ABB RAPID module: Irc6UploadResult.mod

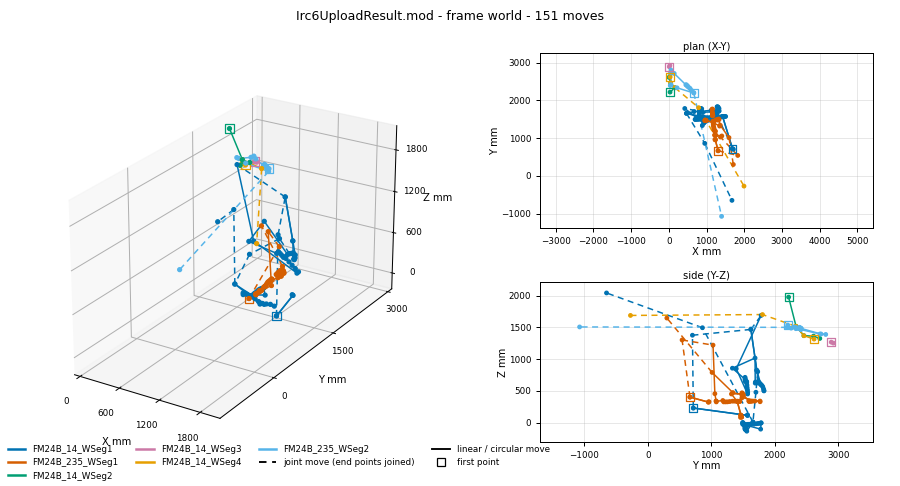
[picture p0: tool path of Irc6UploadResult.mod in frame world, 151 of 155 moves have a stored position in this frame; points joined in program order, loops and branches not executed]
%%%
  VERSION:1
  LANGUAGE:ENGLISH
%%%

MODULE FM24BSegment
!# Process Simulate on eMServer 14 to ABB Rapid Volvo download
!# ------------------------------------------------
!# CREATED   : 26/04/2018 16:18:21 by yogesha
!# CELL      : 2V3 Enginecase_V1
!# ROBOT     : AR21_IRB6700_220-265_SW_IRC5_Grey
!# PROGRAM   : FM24BSegment
!# VOLP      : Abb-Rapid-Volvo 3.14.1
!# RCS       : 6.04.irc5
!# CONTROLLER: 6.0 RW6


!# ----------------------------------------------
!# ------ ROBTARGET
!# ----------------------------------------------
  LOCAL CONST robtarget Towp429210G_10:=[[4329.26,-293.89,1820.66],[0.041749,0.120567,0.991812,0.005418],[-1,0,-1,0],[9e+09,300,9e+09,9e+09,9e+09,9e+09]];
  LOCAL CONST robtarget Towp429210G_20:=[[3458.99,-78.17,1742.31],[0.041752,0.120591,0.991809,0.005444],[0,1,-1,0],[9e+09,25,9e+09,9e+09,9e+09,9e+09]];
  LOCAL CONST robtarget wp429210G:=[[3458.44,-77.54,1729.33],[0.0417533,0.12059,0.991809,0.00543544],[-1,1,-1,0],[9E+09,24.9996,9E+09,9E+09,9E+09,9E+09]];
  LOCAL CONST robtarget Towp431238_10:=[[3458.99,-78.17,1742.31],[0.041752,0.12059,0.991809,0.005444],[0,1,-1,0],[9e+09,25,9e+09,9e+09,9e+09,9e+09]];
  LOCAL CONST robtarget Towp431238_20:=[[4329.31,-293.87,1820.63],[0.041749,0.120567,0.991812,0.005418],[-1,0,-1,0],[9e+09,300,9e+09,9e+09,9e+09,9e+09]];
  LOCAL CONST robtarget Towp431238_30:=[[4344.72,-1189.03,1103.91],[0.199902,-0.332679,-0.8027,-0.452809],[-1,0,-1,0],[9e+09,300,9e+09,9e+09,9e+09,9e+09]];
  LOCAL CONST robtarget Towp431238_40:=[[3393.84,-1017.32,754.57],[0.232734,-0.408546,-0.787878,-0.39771],[0,-1,0,0],[9e+09,200,9e+09,9e+09,9e+09,9e+09]];
  LOCAL CONST robtarget Towp431238_50:=[[3305.21,-568.3,1223.23],[0.212691,-0.544427,-0.755771,-0.295249],[0,-1,0,0],[9e+09,200,9e+09,9e+09,9e+09,9e+09]];
  LOCAL CONST robtarget Towp431238_60:=[[3241.28,-398.98,1372.39],[0.145145,-0.515318,-0.836002,-0.120336],[0,-1,0,0],[9E+09,110.437,9E+09,9E+09,9E+09,9E+09]];
  LOCAL CONST robtarget Towp431238_70:=[[3190.42,-299.46,1405.89],[0.0308017,-0.526819,-0.84797,-0.0495987],[0,0,0,0],[9E+09,44.8475,9E+09,9E+09,9E+09,9E+09]];
  LOCAL CONST robtarget wp431238:=[[3189.5,-297.98,1394.24],[0.030797,-0.526829,-0.847965,-0.049568],[0,0,0,0],[9E+09,24.9996,9E+09,9E+09,9E+09,9E+09]];
  LOCAL CONST robtarget wp429282:=[[3210,-357.62,1373.29],[0.141617,-0.469636,-0.834318,-0.251596],[0,-1,0,0],[9E+09,24.9981,9E+09,9E+09,9E+09,9E+09]];
  LOCAL CONST robtarget wp429283G:=[[3224.18,-374.72,1360.26],[0.231783,-0.536585,-0.744868,-0.321753],[0,-1,0,0],[9E+09,25.0004,9E+09,9E+09,9E+09,9E+09]];
  LOCAL CONST robtarget wp429284:=[[3247.29,-390.89,1343.19],[0.335931,-0.549838,-0.652262,-0.399229],[0,-1,1,0],[9E+09,24.9981,9E+09,9E+09,9E+09,9E+09]];
  LOCAL CONST robtarget wp429285:=[[3274.81,-399.51,1329.50],[0.386439,-0.541317,-0.588631,-0.459515],[0,-1,1,0],[9E+09,24.9999,9E+09,9E+09,9E+09,9E+09]];
  LOCAL CONST robtarget Towp429203G_10:=[[3268.63,-416.83,1335.22],[0.354523,-0.56273,-0.614198,-0.424746],[0,-1,1,0],[9e+09,150,9e+09,9e+09,9e+09,9e+09]];
  LOCAL CONST robtarget Towp429203G_20:=[[3305.16,-568.32,1223.25],[0.212691,-0.544427,-0.755771,-0.295249],[0,-1,0,0],[9e+09,150,9e+09,9e+09,9e+09,9e+09]];
  LOCAL CONST robtarget Towp429203G_30:=[[3393.84,-1017.32,754.57],[0.232734,-0.408546,-0.787878,-0.39771],[0,-1,0,0],[9e+09,150,9e+09,9e+09,9e+09,9e+09]];
  LOCAL CONST robtarget Towp429203G_40:=[[3171.33,-657.72,-21.12],[0.192002,0.140607,-0.823074,0.515668],[0,-1,-2,0],[9e+09,270,9e+09,9e+09,9e+09,9e+09]];
  LOCAL CONST robtarget Towp429203G_50:=[[3598.53,-315.02,877.27],[0.496486,0.441662,-0.526165,0.530647],[0,-1,-2,0],[9e+09,270,9e+09,9e+09,9e+09,9e+09]];
  LOCAL CONST robtarget Towp429203G_60:=[[3461.55,-373.9,1571.05],[0.496488,0.441684,-0.526144,0.530648],[0,-1,-2,0],[9e+09,270,9e+09,9e+09,9e+09,9e+09]];
  LOCAL CONST robtarget wp429203G:=[[3461.52,-406.31,1573.04],[0.496495,0.441685,-0.526141,0.530644],[0,-1,-2,0],[9E+09,24.9993,9E+09,9E+09,9E+09,9E+09]];
  LOCAL CONST robtarget wp429202:=[[3461.25,-404.66,1511.75],[0.423916,0.425319,-0.564527,0.566311],[0,0,-2,0],[9E+09,25.0001,9E+09,9E+09,9E+09,9E+09]];
  LOCAL CONST robtarget wp429201:=[[3462.97,-404.15,1452.61],[0.449062,0.449065,-0.546205,0.546209],[0,-1,-2,0],[9E+09,25.0001,9E+09,9E+09,9E+09,9E+09]];
  LOCAL CONST robtarget wp429200:=[[3463.05,-405.21,1392.26],[0.449062,0.449063,-0.546207,0.546209],[0,-1,-2,0],[9E+09,24.9996,9E+09,9E+09,9E+09,9E+09]];
  LOCAL CONST robtarget wp429199:=[[3463.42,-406.70,1332.03],[0.444279,0.444281,-0.550103,0.550107],[0,-1,-2,0],[9E+09,25.0001,9E+09,9E+09,9E+09,9E+09]];
  LOCAL CONST robtarget wp432680G:=[[3461.83,-405.59,1302.23],[0.407023,0.377506,-0.565637,0.609817],[0,0,-2,0],[9E+09,25.0011,9E+09,9E+09,9E+09,9E+09]];
  LOCAL CONST robtarget wp429273:=[[3482.99,-404.27,1300.72],[0.483124,0.448113,-0.511515,0.551488],[0,0,-2,0],[9E+09,25.0001,9E+09,9E+09,9E+09,9E+09]];
  LOCAL CONST robtarget wp429272:=[[3482.16,-405.26,1268.30],[0.399742,0.399756,-0.583268,0.583267],[0,0,-2,0],[9E+09,24.9996,9E+09,9E+09,9E+09,9E+09]];
  LOCAL CONST robtarget wp429271:=[[3481.99,-406.34,1234.52],[0.399739,0.399755,-0.583271,0.583267],[0,0,-2,0],[9E+09,24.9996,9E+09,9E+09,9E+09,9E+09]];
  LOCAL CONST robtarget wp429270G:=[[3482.14,-406.55,1199.88],[0.373924,0.373932,-0.600148,0.600148],[0,0,-2,0],[9E+09,25.0001,9E+09,9E+09,9E+09,9E+09]];
  LOCAL CONST robtarget Towp429287_10:=[[3479.92,-364.68,1199.99],[0.373918,0.3739,-0.600176,0.600144],[0,0,-2,0],[9e+09,200,9e+09,9e+09,9e+09,9e+09]];
  LOCAL CONST robtarget Towp429287_20:=[[3656.14,-294.7,840.95],[0.373913,0.37388,-0.600196,0.600139],[0,0,-2,0],[9e+09,225,9e+09,9e+09,9e+09,9e+09]];
  LOCAL CONST robtarget Towp429287_30:=[[3301.96,-446.59,772.7],[0.485357,0.438793,-0.503692,0.564078],[0,0,-2,0],[9e+09,100,9e+09,9e+09,9e+09,9e+09]];
  LOCAL CONST robtarget Towp429287_40:=[[3325.47,-372.58,1301.67],[0.485362,0.438786,-0.503693,0.564077],[0,0,-2,0],[9E+09,99.9999,9E+09,9E+09,9E+09,9E+09]];
  LOCAL CONST robtarget wp429287:=[[3324.91,-401.60,1310.54],[0.485353,0.438798,-0.503689,0.564081],[0,0,-2,0],[9E+09,24.9997,9E+09,9E+09,9E+09,9E+09]];
  LOCAL CONST robtarget wp429286:=[[3296.51,-398.64,1318.97],[0.533282,0.418254,-0.478916,0.557955],[0,0,-2,0],[9E+09,24.9994,9E+09,9E+09,9E+09,9E+09]];
  LOCAL CONST robtarget Towp429216G_10:=[[3297.45,-384.27,1310.22],[0.533276,0.418255,-0.478914,0.557961],[0,0,-2,0],[9e+09,100,9e+09,9e+09,9e+09,9e+09]];
  LOCAL CONST robtarget Towp429216G_20:=[[3275.54,-416.71,1074.85],[0.513983,0.427519,-0.492769,0.556981],[0,0,-2,0],[9E+09,100,9E+09,9E+09,9E+09,9E+09]];
  LOCAL CONST robtarget Towp429216G_30:=[[3302.69,609.90,1079.32],[0.491897,0.48192,-0.351229,0.634373],[1,0,-1,0],[9E+09,200,9E+09,9E+09,9E+09,9E+09]];
  LOCAL CONST robtarget Towp429216G_40:=[[3432.85,433.93,1516.60],[0.368379,0.736883,-0.491235,0.282824],[1,-1,-1,0],[9E+09,140.674,9E+09,9E+09,9E+09,9E+09]];
  LOCAL CONST robtarget wp429216G:=[[3460.36,263.26,1671.83],[0.365723,0.756894,-0.437503,0.319295],[1,-1,-1,0],[9E+09,25.0001,9E+09,9E+09,9E+09,9E+09]];
  LOCAL CONST robtarget wp429217:=[[3460.06,290.30,1618.13],[0.33206,0.726093,-0.53763,0.271071],[1,-1,-1,0],[9E+09,24.9996,9E+09,9E+09,9E+09,9E+09]];
  LOCAL CONST robtarget wp429218:=[[3460.14,334.70,1576.96],[0.2765,0.779954,-0.522201,0.206218],[1,-1,-1,0],[9E+09,25.0001,9E+09,9E+09,9E+09,9E+09]];
  LOCAL CONST robtarget wp429219:=[[3461.00,376.35,1534.46],[0.388866,0.719255,-0.497691,0.289411],[1,-1,-1,0],[9E+09,25.0001,9E+09,9E+09,9E+09,9E+09]];
  LOCAL CONST robtarget wp429220G:=[[3462.24,400.89,1481.39],[0.481708,0.646297,-0.461703,0.370253],[1,-1,-1,0],[9E+09,25.0001,9E+09,9E+09,9E+09,9E+09]];
  LOCAL CONST robtarget wp429221:=[[3462.42,411.51,1422.21],[0.547313,0.587418,-0.431084,0.41177],[1,-1,-1,0],[9E+09,25.0001,9E+09,9E+09,9E+09,9E+09]];
  LOCAL CONST robtarget wp429222:=[[3462.28,413.55,1392.21],[0.582433,0.580357,-0.398114,0.40677],[1,-1,-1,0],[9E+09,25.0001,9E+09,9E+09,9E+09,9E+09]];
  LOCAL CONST robtarget wp431518G:=[[3458.41,420.46,1359.28],[0.377325,0.73689,-0.499266,0.255641],[1,-1,-1,0],[9E+09,25.0001,9E+09,9E+09,9E+09,9E+09]];
  LOCAL CONST robtarget wp429263:=[[3481.41,418.56,1361.00],[0.373199,0.728795,-0.510991,0.261665],[1,-1,-1,0],[9E+09,25.0001,9E+09,9E+09,9E+09,9E+09]];
  LOCAL CONST robtarget wp429264:=[[3481.76,433.47,1336.37],[0.467923,0.686198,-0.460136,0.313775],[1,-1,-1,0],[9E+09,25.0001,9E+09,9E+09,9E+09,9E+09]];
  LOCAL CONST robtarget wp429265:=[[3483.02,442.45,1306.90],[0.514146,0.672387,-0.422993,0.32346],[1,-1,-1,0],[9E+09,25.0001,9E+09,9E+09,9E+09,9E+09]];
  LOCAL CONST robtarget wp429266:=[[3481.16,455.69,1277.06],[0.34984,0.757592,-0.500294,0.231024],[1,-1,-1,0],[9E+09,25.0001,9E+09,9E+09,9E+09,9E+09]];
  LOCAL CONST robtarget wp429267G:=[[3480.50,478.18,1255.11],[0.355857,0.777298,-0.471735,0.215962],[1,-1,-1,0],[9E+09,24.9996,9E+09,9E+09,9E+09,9E+09]];
  LOCAL CONST robtarget Towp433102G_10:=[[3479.99,496.17,1270.97],[0.355865,0.777283,-0.471751,0.215968],[1,-1,-1,0],[9e+09,150,9e+09,9e+09,9e+09,9e+09]];
  LOCAL CONST robtarget Towp433102G_20:=[[3211.27,432.33,1467.96],[0.202641,0.500327,-0.809314,0.231561],[1,-1,0,0],[9e+09,130,9e+09,9e+09,9e+09,9e+09]];
  LOCAL CONST robtarget wp433102G:=[[3202.22,373.10,1382.13],[0.131743,0.518539,-0.82381,0.187345],[1,-1,0,0],[9E+09,25.0006,9E+09,9E+09,9E+09,9E+09]];
  LOCAL CONST robtarget Towp429230_10:=[[3202.31,375.23,1386.42],[0.138512,0.516986,-0.822694,0.19161],[1,-1,0,0],[9e+09,25,9e+09,9e+09,9e+09,9e+09]];
  LOCAL CONST robtarget wp429230:=[[3222.80,391.61,1372.68],[0.177635,0.590788,-0.753609,0.226912],[1,-1,0,0],[9E+09,24.9996,9E+09,9E+09,9E+09,9E+09]];
  LOCAL CONST robtarget wp429229:=[[3247.09,402.51,1364.21],[0.258409,0.688458,-0.63409,0.239124],[1,-1,-1,0],[9E+09,25.0001,9E+09,9E+09,9E+09,9E+09]];
  LOCAL CONST robtarget wp429228:=[[3274.77,411.27,1360.35],[0.299271,0.704832,-0.591093,0.25349],[1,-1,-1,0],[9E+09,24.9994,9E+09,9E+09,9E+09,9E+09]];
  LOCAL CONST robtarget wp435330:=[[3311.15,418.41,1362.24],[0.319174,0.778948,-0.441981,0.309873],[1,-1,-1,0],[9E+09,24.9999,9E+09,9E+09,9E+09,9E+09]];
  LOCAL CONST robtarget wp429225:=[[3360.20,420.14,1361.29],[0.37043,0.735721,-0.506434,0.254992],[1,-1,-1,0],[9E+09,25.0001,9E+09,9E+09,9E+09,9E+09]];
  LOCAL CONST robtarget wp429224:=[[3388.55,420.54,1361.74],[0.369194,0.732673,-0.510579,0.257285],[1,-1,-1,0],[9E+09,24.9981,9E+09,9E+09,9E+09,9E+09]];
  LOCAL CONST robtarget wp429223:=[[3418.13,420.96,1362.93],[0.373371,0.733676,-0.505974,0.257495],[1,-1,-1,0],[9E+09,24.9999,9E+09,9E+09,9E+09,9E+09]];
  LOCAL CONST robtarget Frwp429223_10:=[[3419.47,437.29,1376.00],[0.37778,0.742391,-0.493107,0.250966],[1,-1,-1,0],[9E+09,150,9E+09,9E+09,9E+09,9E+09]];
  LOCAL CONST robtarget Frwp429223_20:=[[3302.73,609.92,1079.3],[0.566533,0.521636,-0.288972,0.568711],[1,0,-1,0],[9e+09,200,9e+09,9e+09,9e+09,9e+09]];
  LOCAL CONST robtarget Frwp429223_30:=[[4131.69,-803.62,455.75],[0.261761,0.576711,-0.326948,0.70142],[1,-1,-1,0],[9E+09,330,9E+09,9E+09,9E+09,9E+09]];
  LOCAL CONST robtarget Frwp429223_40:=[[5691.66,-1613.7,572.8],[0.123608,0.891176,-0.221992,0.375828],[0,-1,-2,0],[9e+09,50,9e+09,9e+09,9e+09,9e+09]];
  LOCAL CONST robtarget Towp431451G_10:=[[4354.11,-179.99,1414.82],[0.017246,-0.153263,-0.988031,-0.002663],[-1,0,-1,0],[9e+09,50,9e+09,9e+09,9e+09,9e+09]];
  LOCAL CONST robtarget Towp431451G_20:=[[4058.85,-86.14,1425.65],[0.017246,-0.153263,-0.988031,-0.002663],[-1,0,-1,0],[9e+09,50,9e+09,9e+09,9e+09,9e+09]];
  LOCAL CONST robtarget wp431451G:=[[4047.79,-84.24,1413.94],[0.0172455,-0.153278,-0.988029,-0.00267298],[-1,0,-1,0],[9E+09,24.9999,9E+09,9E+09,9E+09,9E+09]];
  LOCAL CONST robtarget Towp431454_10:=[[4058.85,-86.14,1425.65],[0.017247,-0.153263,-0.988031,-0.002663],[-1,0,-1,0],[9e+09,50,9e+09,9e+09,9e+09,9e+09]];
  LOCAL CONST robtarget Towp431454_20:=[[4354.11,-179.99,1414.82],[0.017247,-0.153263,-0.988031,-0.002663],[-1,0,-1,0],[9e+09,50,9e+09,9e+09,9e+09,9e+09]];
  LOCAL CONST robtarget Towp431454_30:=[[4515.84,-1198.04,1231.54],[0.333428,-0.399022,-0.71079,-0.473693],[-1,0,-1,0],[9e+09,50,9e+09,9e+09,9e+09,9e+09]];
  LOCAL CONST robtarget Towp431454_40:=[[3996.15,-866.5,959.64],[0.272368,-0.516788,-0.761016,-0.282135],[0,-1,0,0],[9e+09,200,9e+09,9e+09,9e+09,9e+09]];
  LOCAL CONST robtarget Towp431454_50:=[[3969.98,-302.77,1478.75],[0.234287,-0.597837,-0.743082,-0.188494],[0,-1,0,0],[9E+09,200,9E+09,9E+09,9E+09,9E+09]];
  LOCAL CONST robtarget Towp431454_60:=[[3939.13,-116.51,1431.85],[0.026894,-0.626479,-0.778673,-0.021648],[0,0,0,0],[9E+09,66.9781,9E+09,9E+09,9E+09,9E+09]];
  LOCAL CONST robtarget wp431454:=[[3932.99,-80.90,1413.88],[8.26877E-07,0.626854,0.779136,-2.96273E-06],[0,0,0,0],[9E+09,24.9999,9E+09,9E+09,9E+09,9E+09]];
  LOCAL CONST robtarget Towp431457_10:=[[3937.3,-102.5,1425.97],[0.000001,0.626851,0.779139,0.000001],[0,0,0,0],[9e+09,50,9e+09,9e+09,9e+09,9e+09]];
  LOCAL CONST robtarget Towp431457_20:=[[3832.32,-119.5,1426.02],[1E-06,0.543807,0.83921,1E-06],[0,0,0,0],[9E+09,50,9E+09,9E+09,9E+09,9E+09]];
  LOCAL CONST robtarget wp431457:=[[3816.00,-81.56,1414.18],[1.15086E-06,0.543808,0.83921,-2.43318E-06],[0,0,0,0],[9E+09,24.9999,9E+09,9E+09,9E+09,9E+09]];
  LOCAL CONST robtarget wp431458:=[[3786.49,-81.08,1414.19],[3.84991E-06,0.519799,0.854289,-2.12541E-06],[0,0,0,0],[9E+09,25.0004,9E+09,9E+09,9E+09,9E+09]];
  LOCAL CONST robtarget wp432845:=[[3756.45,-81.29,1412.87],[0.0450299,0.604524,0.794575,0.0342574],[0,0,0,0],[9E+09,24.9999,9E+09,9E+09,9E+09,9E+09]];
  LOCAL CONST robtarget wp432844G:=[[3720.23,-81.36,1405.62],[0.103024,0.598136,0.790917,0.0779127],[0,0,0,0],[9E+09,24.9999,9E+09,9E+09,9E+09,9E+09]];
  LOCAL CONST robtarget wp431461:=[[3676.01,-81.72,1397.15],[1.83255E-06,0.474376,0.880323,-1.16515E-05],[0,0,0,0],[9E+09,24.9994,9E+09,9E+09,9E+09,9E+09]];
  LOCAL CONST robtarget wp431462:=[[3641.72,-81.95,1396.93],[2.5744E-07,0.453114,0.891453,-1.06155E-06],[0,0,0,0],[9E+09,24.9999,9E+09,9E+09,9E+09,9E+09]];
  LOCAL CONST robtarget wp431463:=[[3601.74,-82.52,1396.64],[5.1017E-06,0.411813,0.911268,-4.07155E-06],[0,0,0,0],[9E+09,24.9999,9E+09,9E+09,9E+09,9E+09]];
  LOCAL CONST robtarget wp431464:=[[3561.70,-82.58,1394.92],[7.74193E-06,0.377741,0.925911,-1.0349E-05],[0,0,0,0],[9E+09,24.9999,9E+09,9E+09,9E+09,9E+09]];
  LOCAL CONST robtarget Towp432811G_10:=[[3561.65,-83.01,1407.42],[0.000002,0.377731,0.925915,0.000001],[0,0,0,0],[9e+09,50,9e+09,9e+09,9e+09,9e+09]];
  LOCAL CONST robtarget Towp432811G_20:=[[3601.71,-82.98,1408.41],[0.000002,0.411804,0.911273,0.000001],[0,0,0,0],[9e+09,25,9e+09,9e+09,9e+09,9e+09]];
  LOCAL CONST robtarget Towp432811G_30:=[[3516.22,241.86,1399.88],[0.029328,-0.541645,-0.839883,-0.018915],[0,0,0,0],[9e+09,50,9e+09,9e+09,9e+09,9e+09]];
  LOCAL CONST robtarget wp432811G:=[[3533.56,253.42,1393.93],[0.00291459,-0.549291,-0.835624,-0.00191196],[0,0,0,0],[9E+09,25.0004,9E+09,9E+09,9E+09,9E+09]];
  LOCAL CONST robtarget Towp432812G_10:=[[3516.27,241.87,1399.86],[0.029328,-0.541645,-0.839883,-0.018915],[0,0,0,0],[9e+09,50,9e+09,9e+09,9e+09,9e+09]];
  LOCAL CONST robtarget Towp432812G_20:=[[3529.9,204.56,1398.89],[0.014868,-0.523433,-0.851888,-0.009137],[0,0,0,0],[9e+09,25,9e+09,9e+09,9e+09,9e+09]];
  LOCAL CONST robtarget wp432812G:=[[3533.86,207.53,1393.12],[3.79802E-06,0.523518,0.852015,-2.18588E-06],[0,0,0,0],[9E+09,25,9E+09,9E+09,9E+09,9E+09]];
  LOCAL CONST robtarget Towp432815G_10:=[[3529.9,204.56,1398.89],[0.014868,-0.523433,-0.851888,-0.009137],[0,0,0,0],[9e+09,25,9e+09,9e+09,9e+09,9e+09]];
  LOCAL CONST robtarget Towp432815G_20:=[[3601.71,-82.98,1408.4],[0.000002,0.411804,0.911273,0.000001],[0,0,0,0],[9e+09,300,9e+09,9e+09,9e+09,9e+09]];
  LOCAL CONST robtarget Towp432815G_30:=[[3705.12,-274.41,1451.67],[5.86579E-06,0.419365,0.907818,6.25013E-06],[0,0,0,0],[9E+09,300.001,9E+09,9E+09,9E+09,9E+09]];
  LOCAL CONST robtarget Towp432815G_40:=[[3529.15,-277.66,1446.44],[1.07647E-05,0.329276,0.944234,-2.33319E-06],[0,0,0,0],[9E+09,300,9E+09,9E+09,9E+09,9E+09]];
  LOCAL CONST robtarget Towp432815G_50:=[[3533.49,-249.64,1410.91],[0.000002,0.318433,0.947945,0.000001],[0,0,0,0],[9e+09,300,9e+09,9e+09,9e+09,9e+09]];
  LOCAL CONST robtarget wp432815G:=[[3533.51,-249.64,1392.73],[3.23588E-07,-0.318437,-0.947944,-6.32931E-07],[0,0,0,0],[9E+09,25,9E+09,9E+09,9E+09,9E+09]];
  LOCAL CONST robtarget Towp432814G_10:=[[3533.49,-249.64,1445.91],[0.000002,0.318433,0.947945,0.000001],[0,0,0,0],[9e+09,300,9e+09,9e+09,9e+09,9e+09]];
  LOCAL CONST robtarget Towp432814G_20:=[[3533.54,-206.31,1455.89],[0.000002,0.425672,0.904877,0.000001],[0,0,0,0],[9e+09,300,9e+09,9e+09,9e+09,9e+09]];
  LOCAL CONST robtarget wp432814G:=[[3533.51,-206.32,1393.52],[6.70131E-06,0.425675,0.904876,-3.17874E-06],[0,0,0,0],[9E+09,25,9E+09,9E+09,9E+09,9E+09]];
  LOCAL CONST robtarget Towp431473_10:=[[3533.53,-206.31,1455.88],[0.000002,0.41776,0.908558,0.000001],[0,0,0,0],[9e+09,300,9e+09,9e+09,9e+09,9e+09]];
  LOCAL CONST robtarget Towp431473_20:=[[3241.66,-83.02,1412.41],[6.10042E-06,0.306933,0.951731,1.0367E-05],[0,0,0,0],[9E+09,100,9E+09,9E+09,9E+09,9E+09]];
  LOCAL CONST robtarget wp431473:=[[3241.66,-81.77,1393.96],[1.3303E-05,0.30694,0.951729,3.48439E-06],[0,0,0,0],[9E+09,24.9999,9E+09,9E+09,9E+09,9E+09]];
  LOCAL CONST robtarget wp431471:=[[3321.74,-82.92,1396.00],[3.51303E-06,0.35415,0.935189,-8.41567E-06],[0,0,0,0],[9E+09,25.0004,9E+09,9E+09,9E+09,9E+09]];
  LOCAL CONST robtarget wp431470:=[[3355.01,-82.96,1396.34],[4.77567E-06,0.375719,0.926734,-5.52436E-06],[0,0,0,0],[9E+09,24.9999,9E+09,9E+09,9E+09,9E+09]];
  LOCAL CONST robtarget wp431469:=[[3381.69,-82.96,1395.83],[4.98806E-06,0.381775,0.924255,-4.33881E-06],[0,0,0,0],[9E+09,25.0004,9E+09,9E+09,9E+09,9E+09]];
  LOCAL CONST robtarget Towp431468G_10:=[[3384.98,-83,1402.43],[1E-06,0.381768,0.924258,1E-06],[0,0,0,0],[9E+09,30,9E+09,9E+09,9E+09,9E+09]];
  LOCAL CONST robtarget Towp431468G_20:=[[3414.26,-83,1403.43],[4.22424E-06,0.425982,0.904731,7.73845E-06],[0,0,0,0],[9E+09,30,9E+09,9E+09,9E+09,9E+09]];
  LOCAL CONST robtarget wp431468G:=[[3417.52,-83.00,1387.95],[2.74018E-06,0.425977,0.904734,-2.87824E-06],[0,0,0,0],[9E+09,24.9999,9E+09,9E+09,9E+09,9E+09]];
  LOCAL CONST robtarget Frwp431468G_10:=[[3412.65,-83.00,1403.44],[1.85513E-06,0.425983,0.904731,5.85803E-06],[0,0,0,0],[9E+09,200,9E+09,9E+09,9E+09,9E+09]];
  LOCAL CONST robtarget Frwp431468G_20:=[[3514.45,-256.52,1454.18],[2.55326E-06,0.318434,0.947945,2.20187E-06],[0,0,0,0],[9E+09,300,9E+09,9E+09,9E+09,9E+09]];
  LOCAL CONST robtarget Frwp431468G_30:=[[3684.45,-303.36,1451.55],[2.68411E-05,0.356372,0.934344,-9.8449E-06],[0,0,0,0],[9E+09,300,9E+09,9E+09,9E+09,9E+09]];
  LOCAL CONST robtarget Frwp431468G_40:=[[4027.69,-679.08,1407.41],[0.000002,0.295595,0.955313,0.000001],[-1,0,0,0],[9e+09,300,9e+09,9e+09,9e+09,9e+09]];
  LOCAL CONST robtarget Frwp431468G_50:=[[4746.66,-1377.99,907.35],[0.224016,-0.67974,-0.349694,-0.604553],[-1,0,-1,0],[9E+09,50.0009,9E+09,9E+09,9E+09,9E+09]];
  LOCAL CONST robtarget Towp433113_10:=[[3347.95,834.06,944.48],[0.127353,-0.51805,0.839702,0.101518],[0,0,-3,0],[9E+09,242,9E+09,9E+09,9E+09,9E+09]];
  LOCAL CONST robtarget Towp433113_20:=[[3426.57,520.61,1315.50],[0.184335,-0.578607,0.784932,-0.122949],[0,0,-2,0],[9E+09,242.273,9E+09,9E+09,9E+09,9E+09]];
  LOCAL CONST robtarget Towp433113_30:=[[3274.99,407.19,1434.32],[0.0363408,-0.545988,0.805467,-0.227594],[0,0,-2,0],[9E+09,242.273,9E+09,9E+09,9E+09,9E+09]];
  LOCAL CONST robtarget wp433113:=[[3170.31,293.40,1400.96],[1.26895E-05,0.520754,-0.853707,-1.23285E-06],[0,0,-3,0],[9E+09,25.0004,9E+09,9E+09,9E+09,9E+09]];
  LOCAL CONST robtarget wp433110:=[[3168.72,179.18,1396.97],[1.02956E-05,0.6106,-0.791939,1.47874E-06],[1,-1,-2,0],[9E+09,24.9958,9E+09,9E+09,9E+09,9E+09]];
  LOCAL CONST robtarget wp432852:=[[3060.10,20.02,1401.72],[0.0278666,0.601599,-0.798036,-0.0210104],[1,-1,-2,0],[9E+09,25,9E+09,9E+09,9E+09,9E+09]];
  LOCAL CONST robtarget wp432849:=[[3060.15,-19.99,1402.41],[0.027635,0.610267,-0.791426,-0.021315],[1,-1,-2,0],[9e+09,25,9e+09,9e+09,9e+09,9e+09]];
  LOCAL CONST robtarget Frwp432849_10:=[[3195.54,257.28,1437.13],[0.0242642,-0.583135,0.797611,-0.152251],[0,0,-2,0],[9E+09,169.434,9E+09,9E+09,9E+09,9E+09]];
  LOCAL CONST robtarget Frwp432849_20:=[[3275.00,407.18,1434.33],[0.0363405,-0.545991,0.805465,-0.227594],[0,0,-2,0],[9E+09,242.273,9E+09,9E+09,9E+09,9E+09]];
  LOCAL CONST robtarget Frwp432849_30:=[[3426.57,520.60,1315.50],[0.184333,-0.578608,0.784932,-0.122949],[0,0,-2,0],[9E+09,242.273,9E+09,9E+09,9E+09,9E+09]];
  LOCAL CONST robtarget Frwp432849_40:=[[3319.21,549.75,1278.15],[0.00613,-0.582455,0.812824,0.005057],[1,0,-2,0],[9e+09,290,9e+09,9e+09,9e+09,9e+09]];
  LOCAL CONST robtarget Frwp432849_50:=[[4215.11,789.08,1199.66],[0.410336,-0.68266,0.516184,-0.314887],[0,0,-2,0],[9E+09,10.0002,9E+09,9E+09,9E+09,9E+09]];
  LOCAL CONST robtarget Frwp432849_60:=[[6189.98,2078.47,1654.43],[0.626281,-0.760132,-0.0766629,-0.155224],[0,0,-2,0],[9E+09,10.0002,9E+09,9E+09,9E+09,9E+09]];
  LOCAL CONST robtarget Towp431452_20:=[[4144.33,-76.09,1416.25],[0.00083,-0.543594,0.839346,-0.001624],[1,-1,-2,0],[9e+09,75,9e+09,9e+09,9e+09,9e+09]];
  LOCAL CONST robtarget Towp431452_30:=[[4060.20,-83.00,1449.04],[4.52795E-06,0.542918,-0.839786,6.62105E-07],[0,-1,-2,0],[9E+09,77.7032,9E+09,9E+09,9E+09,9E+09]];
  LOCAL CONST robtarget wp431452:=[[3997.78,-86.85,1420.63],[5.21495E-06,0.542922,-0.839783,-1.50726E-06],[1,-1,-2,0],[9E+09,24.9996,9E+09,9E+09,9E+09,9E+09]];
  LOCAL CONST robtarget wp431453:=[[3964.42,-87.19,1419.54],[1.90782E-06,-0.610601,0.791939,-1.82666E-06],[1,-1,-2,0],[9E+09,25.0001,9E+09,9E+09,9E+09,9E+09]];
  LOCAL CONST robtarget Towp432847_10:=[[3909.15,-83.03,1425.96],[4.58738E-06,0.570119,-0.821562,-5.22273E-06],[1,-1,-2,0],[9E+09,24.9999,9E+09,9E+09,9E+09,9E+09]];
  LOCAL CONST robtarget wp432847:=[[3894.80,-87.57,1411.16],[5.75398E-07,-0.559311,0.828958,1.97935E-06],[1,-1,-2,0],[9E+09,25.0001,9E+09,9E+09,9E+09,9E+09]];
  LOCAL CONST robtarget wp432846:=[[3853.51,-88.16,1411.04],[1.09929E-05,-0.557497,0.830179,-1.38076E-07],[1,-1,-2,0],[9E+09,25.0001,9E+09,9E+09,9E+09,9E+09]];
  LOCAL CONST robtarget Towp431472_10:=[[3839.99,-83.03,1431.31],[8.35906E-06,-0.554335,0.832294,5.97258E-06],[1,-1,-2,0],[9E+09,38.6234,9E+09,9E+09,9E+09,9E+09]];
  LOCAL CONST robtarget Towp431472_20:=[[3404.30,-84.22,1417.84],[7.11336E-06,0.463168,-0.88627,-5.6972E-06],[1,-1,-2,0],[9E+09,38.9197,9E+09,9E+09,9E+09,9E+09]];
  LOCAL CONST robtarget wp431472:=[[3280.55,-86.11,1400.95],[1.56873E-05,-0.436537,0.899686,-9.90722E-07],[1,-1,-2,0],[9E+09,24.9996,9E+09,9E+09,9E+09,9E+09]];
  LOCAL CONST robtarget Towp432810_10:=[[3332.04,-33.93,1413.54],[2.18771E-06,0.439395,-0.898294,1.92756E-06],[1,-1,-2,0],[9E+09,40.0521,9E+09,9E+09,9E+09,9E+09]];
  LOCAL CONST robtarget Towp432810_20:=[[3559.46,195.02,1409.03],[2.09E-06,0.452279,-0.891877,3.27153E-06],[1,-1,-2,0],[9E+09,38.4337,9E+09,9E+09,9E+09,9E+09]];
  LOCAL CONST robtarget wp432810:=[[3567.15,227.98,1398.05],[1.87051E-05,0.454113,-0.890944,7.4278E-07],[1,-1,-2,0],[9E+09,25,9E+09,9E+09,9E+09,9E+09]];
  LOCAL CONST robtarget Frwp432810_10:=[[3730.79,138.86,1435.88],[0.000936145,-0.480398,0.877049,-0.00151362],[1,-1,-2,0],[9E+09,57.0615,9E+09,9E+09,9E+09,9E+09]];
  LOCAL CONST robtarget Frwp432810_20:=[[4144.37,-76.10,1454.50],[0.000826724,-0.543602,0.839341,-0.00162357],[0,-1,-2,0],[9E+09,75.0001,9E+09,9E+09,9E+09,9E+09]];
  LOCAL CONST robtarget Frwp432810_30:=[[6890.16,1648.41,2297.46],[0.547499,-0.703355,-0.392109,-0.227569],[0,-1,-1,0],[9E+09,75.0006,9E+09,9E+09,9E+09,9E+09]];


!# -----------------------------------------------
!# ------ SPOT DATA
!# -----------------------------------------------

  LOCAL PERS spotdata sd_wp429210:=[429210,1,1,1];
  LOCAL PERS spotdata sd_wp431238:=[431238,1,1,1];
  LOCAL PERS spotdata sd_wp429282:=[429282,1,1,1];
  LOCAL PERS spotdata sd_wp429283:=[429283,1,1,1];
  LOCAL PERS spotdata sd_wp429284:=[429284,1,1,1];
  LOCAL PERS spotdata sd_wp429285:=[429285,1,1,1];
  LOCAL PERS spotdata sd_wp429203:=[429203,1,1,1];
  LOCAL PERS spotdata sd_wp429202:=[429202,1,1,1];
  LOCAL PERS spotdata sd_wp429201:=[429201,1,1,1];
  LOCAL PERS spotdata sd_wp429200:=[429200,1,1,1];
  LOCAL PERS spotdata sd_wp429199:=[429199,1,1,1];
  LOCAL PERS spotdata sd_wp432680:=[432680,1,1,1];
  LOCAL PERS spotdata sd_wp429273:=[429273,1,1,1];
  LOCAL PERS spotdata sd_wp429272:=[429272,1,1,1];
  LOCAL PERS spotdata sd_wp429271:=[429271,1,1,1];
  LOCAL PERS spotdata sd_wp429270:=[429270,1,1,1];
  LOCAL PERS spotdata sd_wp429267:=[429267,1,1,1];
  LOCAL PERS spotdata sd_wp429287:=[429287,1,1,1];
  LOCAL PERS spotdata sd_wp429286:=[429286,1,1,1];
  LOCAL PERS spotdata sd_wp429216:=[429216,1,1,1];
  LOCAL PERS spotdata sd_wp429217:=[429217,1,1,1];
  LOCAL PERS spotdata sd_wp429218:=[429218,1,1,1];
  LOCAL PERS spotdata sd_wp429219:=[429219,1,1,1];
  LOCAL PERS spotdata sd_wp429220:=[429220,1,1,1];
  LOCAL PERS spotdata sd_wp429221:=[429221,1,1,1];
  LOCAL PERS spotdata sd_wp429222:=[429222,1,1,1];
  LOCAL PERS spotdata sd_wp431518:=[431518,1,1,1];
  LOCAL PERS spotdata sd_wp429263:=[429263,1,1,1];
  LOCAL PERS spotdata sd_wp429264:=[429264,1,1,1];
  LOCAL PERS spotdata sd_wp429265:=[429265,1,1,1];
  LOCAL PERS spotdata sd_wp429266:=[429266,1,1,1];
  LOCAL PERS spotdata sd_wp433102:=[433102,1,1,1];
  LOCAL PERS spotdata sd_wp429230:=[429230,1,1,1];
  LOCAL PERS spotdata sd_wp429229:=[429229,1,1,1];
  LOCAL PERS spotdata sd_wp429228:=[429228,1,1,1];
  LOCAL PERS spotdata sd_wp435330:=[435330,1,1,1];
  LOCAL PERS spotdata sd_wp429225:=[429225,1,1,1];
  LOCAL PERS spotdata sd_wp429224:=[429224,1,1,1];
  LOCAL PERS spotdata sd_wp429223:=[429223,1,1,1];
  LOCAL PERS spotdata sd_wp431451:=[431451,1,1,1];
  LOCAL PERS spotdata sd_wp431454:=[431454,1,1,1];
  LOCAL PERS spotdata sd_wp431457:=[431457,1,1,1];
  LOCAL PERS spotdata sd_wp431458:=[431458,1,1,1];
  LOCAL PERS spotdata sd_wp432845:=[432845,1,1,1];
  LOCAL PERS spotdata sd_wp432844:=[432844,1,1,1];
  LOCAL PERS spotdata sd_wp431461:=[431461,1,1,1];
  LOCAL PERS spotdata sd_wp431462:=[431462,1,1,1];
  LOCAL PERS spotdata sd_wp431463:=[431463,1,1,1];
  LOCAL PERS spotdata sd_wp431464:=[431464,1,1,1];
  LOCAL PERS spotdata sd_wp432811:=[432811,1,1,1];
  LOCAL PERS spotdata sd_wp432812:=[432812,1,1,1];
  LOCAL PERS spotdata sd_wp432815:=[432815,1,1,1];
  LOCAL PERS spotdata sd_wp432814:=[432814,1,1,1];
  LOCAL PERS spotdata sd_wp431473:=[431473,1,1,1];
  LOCAL PERS spotdata sd_wp431471:=[431471,1,1,1];
  LOCAL PERS spotdata sd_wp431470:=[431470,1,1,1];
  LOCAL PERS spotdata sd_wp431469:=[431469,1,1,1];
  LOCAL PERS spotdata sd_wp431468:=[431468,1,1,1];
  LOCAL PERS spotdata sd_wp433113:=[433113,1,1,1];
  LOCAL PERS spotdata sd_wp433110:=[433110,1,1,1];
  LOCAL PERS spotdata sd_wp432852:=[432852,1,1,1];
  LOCAL PERS spotdata sd_wp432849:=[432849,1,1,1];
  LOCAL PERS spotdata sd_wp431452:=[431452,1,1,1];
  LOCAL PERS spotdata sd_wp431453:=[431453,1,1,1];
  LOCAL PERS spotdata sd_wp432847:=[432847,1,1,1];
  LOCAL PERS spotdata sd_wp432846:=[432846,1,1,1];
  LOCAL PERS spotdata sd_wp431472:=[431472,1,1,1];
  LOCAL PERS spotdata sd_wp432810:=[432810,1,1,1];

!# -----------------------------------------------
!# ------ WOBJ DATA
!# -----------------------------------------------
  PERS wobjdata wFM24B_Cabframe:=[FALSE,TRUE,"""",[[-212.9,4917.65,1167.66],[-0.310964,0.663413,-0.616213,0.288904]],[[0,0,0],[1,0,0,0]]];
  PERS wobjdata wFM24B_CabframeUQ53:=[FALSE,TRUE,"""",[[-210.08,4920.13,1168.24],[-0.310764,0.6630223,-0.6166411,0.2891035]],[[0,0,0],[1,0,0,0]]];
  PERS wobjdata wFM24B_CabframeUQ54:=[FALSE,TRUE,"""",[[-212.9,4917.65,1167.66],[-0.3109636,0.6634134,-0.6162131,0.2889042]],[[0,0,0],[1,0,0,0]]];
  PERS wobjdata wFM24BL1_CabframeGrip:=[FALSE,TRUE,"""",[[-2504.52,4649.77,2641.4],[0.1735002,0.9601499,-0.2131685,-0.0506865]],[[0,0,0],[1,0,0,0]]];
  PERS wobjdata wFM24BL2_CabframeGrip:=[FALSE,TRUE,"""",[[-2337.92,5336.45,2143],[0.1189337,0.9166429,-0.3778935,0.0530758]],[[0,0,0],[1,0,0,0]]];
  LOCAL CONST robtarget wp431248:=[[3198.54,-334.59,1396.68],[0.0870968,-0.499441,-0.84835,-0.152561],[0,0,0,0],[9E+09,24.9997,9E+09,9E+09,9E+09,9E+09]];
  LOCAL CONST robtarget wp429238:=[[3460.25,366.29,1559.70],[0.340751,0.747978,-0.5099,0.25381],[1,-1,-1,0],[9E+09,24.9996,9E+09,9E+09,9E+09,9E+09]];
  LOCAL CONST robtarget wp429239:=[[3461.35,397.68,1509.44],[0.439763,0.682037,-0.479726,0.333613],[1,-1,-1,0],[9E+09,24.9996,9E+09,9E+09,9E+09,9E+09]];
  LOCAL CONST robtarget Towp429216G_50:=[[3271.02,117.74,936.91],[0.454928,0.442573,-0.429627,0.642332],[0,0,-2,0],[9E+09,159.596,9E+09,9E+09,9E+09,9E+09]];
PERS spotdata spot_testweld:=[195,0,0,0];

  PROC FM24B_14_WSeg1()
     MoveAbsJ HomeXQ11Gun,v2500,fine,XQ11GunTCP;
     MoveJ Towp429210G_10,v2500,z200,XQ11GunTCP\Wobj:=wFM24B_Cabframe;
     MoveL Towp429210G_20,v2500,z50,XQ11GunTCP\Wobj:=wFM24B_Cabframe;
     SpotL wp429210G,v2500,sd_wp429210,XQ11Gun\GunD:=XQ11GunData,XQ11GunTCP\Wobj:=wFM24B_Cabframe;
     MoveL Towp431238_10,v2500,z50,XQ11GunTCP\Wobj:=wFM24B_Cabframe;
     MoveL Towp431238_20,v2500,z50,XQ11GunTCP\Wobj:=wFM24B_Cabframe;
     MoveJ Towp431238_30,v2500,z50,XQ11GunTCP\Wobj:=wFM24B_Cabframe;
     MoveJ Towp431238_40,v2500,z50,XQ11GunTCP\Wobj:=wFM24B_Cabframe;
     MoveL Towp431238_50,v2500,z50,XQ11GunTCP\Wobj:=wFM24B_Cabframe;
     MoveL Towp431238_60,v2500,z50,XQ11GunTCP\Wobj:=wFM24B_Cabframe;
     MoveL Towp431238_70,v2500,z50,XQ11GunTCP\Wobj:=wFM24B_Cabframe;
     SpotL wp431238,v2500,sd_wp431238,XQ11Gun\GunD:=XQ11GunData,XQ11GunTCP\Wobj:=wFM24B_Cabframe;
     MoveL wp431248, v2500, z100, XQ11GunTCP\WObj:=wFM24B_Cabframe;
     SpotL wp429282,v2500,sd_wp429282,XQ11Gun\GunD:=XQ11GunData,XQ11GunTCP\Wobj:=wFM24B_Cabframe;
     SpotL wp429283G,v2500,sd_wp429283,XQ11Gun\GunD:=XQ11GunData,XQ11GunTCP\Wobj:=wFM24B_Cabframe;
     SpotL wp429284,v2500,sd_wp429284,XQ11Gun\GunD:=XQ11GunData,XQ11GunTCP\Wobj:=wFM24B_Cabframe;
     SpotL wp429285,v2500,sd_wp429285,XQ11Gun\GunD:=XQ11GunData,XQ11GunTCP\Wobj:=wFM24B_Cabframe;
     MoveL Towp429203G_10,v2500,z50,XQ11GunTCP\Wobj:=wFM24B_Cabframe;
     MoveL Towp429203G_20,v2500,z50,XQ11GunTCP\Wobj:=wFM24B_Cabframe;
     MoveL Towp429203G_30,v2500,z50,XQ11GunTCP\Wobj:=wFM24B_Cabframe;
     MoveJ Towp429203G_40,v2500,z50,XQ11GunTCP\Wobj:=wFM24B_Cabframe;
     MoveL Towp429203G_50,v2500,z50,XQ11GunTCP\Wobj:=wFM24B_Cabframe;
     MoveL Towp429203G_60,v2500,z50,XQ11GunTCP\Wobj:=wFM24B_Cabframe;
     SpotL wp429203G,v2500,sd_wp429203,XQ11Gun\GunD:=XQ11GunData,XQ11GunTCP\Wobj:=wFM24B_Cabframe;
     SpotL wp429202,v2500,sd_wp429202,XQ11Gun\GunD:=XQ11GunData,XQ11GunTCP\Wobj:=wFM24B_Cabframe;
     SpotL wp429201,v2500,sd_wp429201,XQ11Gun\GunD:=XQ11GunData,XQ11GunTCP\Wobj:=wFM24B_Cabframe;
     SpotL wp429200,v2500,sd_wp429200,XQ11Gun\GunD:=XQ11GunData,XQ11GunTCP\Wobj:=wFM24B_Cabframe;
     SpotL wp429199,v2500,sd_wp429199,XQ11Gun\GunD:=XQ11GunData,XQ11GunTCP\Wobj:=wFM24B_Cabframe;
     SpotL wp432680G,v2500,sd_wp432680,XQ11Gun\GunD:=XQ11GunData,XQ11GunTCP\Wobj:=wFM24B_Cabframe;
     SpotL wp429273,v2500,sd_wp429273,XQ11Gun\GunD:=XQ11GunData,XQ11GunTCP\Wobj:=wFM24B_Cabframe;
     SpotL wp429272,v2500,sd_wp429272,XQ11Gun\GunD:=XQ11GunData,XQ11GunTCP\Wobj:=wFM24B_Cabframe;
     SpotL wp429271,v2500,sd_wp429271,XQ11Gun\GunD:=XQ11GunData,XQ11GunTCP\Wobj:=wFM24B_Cabframe;
     SpotL wp429270G,v2500,sd_wp429270,XQ11Gun\GunD:=XQ11GunData,XQ11GunTCP\Wobj:=wFM24B_Cabframe;
     MoveL Towp429287_10,v2500,z50,XQ11GunTCP\Wobj:=wFM24B_Cabframe;
     MoveL Towp429287_20,v2500,z50,XQ11GunTCP\Wobj:=wFM24B_Cabframe;
     MoveL Towp429287_30,v2500,z50,XQ11GunTCP\Wobj:=wFM24B_Cabframe;
     MoveL Towp429287_40,v2500,z50,XQ11GunTCP\Wobj:=wFM24B_Cabframe;
     SpotL wp429287,v2500,sd_wp429287,XQ11Gun\GunD:=XQ11GunData,XQ11GunTCP\Wobj:=wFM24B_Cabframe;
     SpotL wp429286,v2500,sd_wp429286,XQ11Gun\GunD:=XQ11GunData,XQ11GunTCP\Wobj:=wFM24B_Cabframe;
     MoveL Towp429216G_10,v2500,z50,XQ11GunTCP\Wobj:=wFM24B_Cabframe;
     MoveJ Towp429216G_20,v2500,z50,XQ11GunTCP\Wobj:=wFM24B_Cabframe;
     MoveJ Towp429216G_50, v2500, z50, XQ11GunTCP\WObj:=wFM24B_Cabframe;
     MoveJ Towp429216G_30,v2500,z50,XQ11GunTCP\Wobj:=wFM24B_Cabframe;
     MoveL Towp429216G_40,v2500,z50,XQ11GunTCP\Wobj:=wFM24B_Cabframe;
     SpotL wp429216G,v2500,sd_wp429216,XQ11Gun\GunD:=XQ11GunData,XQ11GunTCP\Wobj:=wFM24B_Cabframe;
     SpotL wp429217,v2500,sd_wp429217,XQ11Gun\GunD:=XQ11GunData,XQ11GunTCP\Wobj:=wFM24B_Cabframe;
     SpotL wp429218,v2500,sd_wp429218,XQ11Gun\GunD:=XQ11GunData,XQ11GunTCP\Wobj:=wFM24B_Cabframe;
     MoveL wp429238, v2500, z50, XQ11GunTCP\WObj:=wFM24B_Cabframe;
     SpotL wp429219,v2500,sd_wp429219,XQ11Gun\GunD:=XQ11GunData,XQ11GunTCP\Wobj:=wFM24B_Cabframe;
     MoveL wp429239, v2500, z50, XQ11GunTCP\WObj:=wFM24B_Cabframe;
     SpotL wp429220G,v2500,sd_wp429220,XQ11Gun\GunD:=XQ11GunData,XQ11GunTCP\Wobj:=wFM24B_Cabframe;
     SpotL wp429221,v2500,sd_wp429221,XQ11Gun\GunD:=XQ11GunData,XQ11GunTCP\Wobj:=wFM24B_Cabframe;
     SpotL wp429222,v2500,sd_wp429222,XQ11Gun\GunD:=XQ11GunData,XQ11GunTCP\Wobj:=wFM24B_Cabframe;
     SpotL wp431518G,v2500,sd_wp431518,XQ11Gun\GunD:=XQ11GunData,XQ11GunTCP\Wobj:=wFM24B_Cabframe;
     SpotL wp429263,v2500,sd_wp429263,XQ11Gun\GunD:=XQ11GunData,XQ11GunTCP\Wobj:=wFM24B_Cabframe;
     SpotL wp429264,v2500,sd_wp429264,XQ11Gun\GunD:=XQ11GunData,XQ11GunTCP\Wobj:=wFM24B_Cabframe;
     SpotL wp429265,v2500,sd_wp429265,XQ11Gun\GunD:=XQ11GunData,XQ11GunTCP\Wobj:=wFM24B_Cabframe;
     SpotL wp429266,v2500,sd_wp429266,XQ11Gun\GunD:=XQ11GunData,XQ11GunTCP\Wobj:=wFM24B_Cabframe;
     SpotL wp429267G,v2500,sd_wp429267,XQ11Gun\GunD:=XQ11GunData,XQ11GunTCP\Wobj:=wFM24B_Cabframe;
     MoveL Towp433102G_10,v2500,z50,XQ11GunTCP\Wobj:=wFM24B_Cabframe;
     MoveL Towp433102G_20,v2500,z50,XQ11GunTCP\Wobj:=wFM24B_Cabframe;
     SpotL wp433102G,v2500,sd_wp433102,XQ11Gun\GunD:=XQ11GunData,XQ11GunTCP\Wobj:=wFM24B_Cabframe;
     MoveL Towp429230_10,v2500,z50,XQ11GunTCP\Wobj:=wFM24B_Cabframe;
     SpotL wp429230,v2500,sd_wp429230,XQ11Gun\GunD:=XQ11GunData,XQ11GunTCP\Wobj:=wFM24B_Cabframe;
     SpotL wp429229,v2500,sd_wp429229,XQ11Gun\GunD:=XQ11GunData,XQ11GunTCP\Wobj:=wFM24B_Cabframe;
     SpotL wp429228,v2500,sd_wp429228,XQ11Gun\GunD:=XQ11GunData,XQ11GunTCP\Wobj:=wFM24B_Cabframe;
     SpotL wp435330,v2500,sd_wp435330,XQ11Gun\GunD:=XQ11GunData,XQ11GunTCP\Wobj:=wFM24B_Cabframe;
     SpotL wp429225,v2500,sd_wp429225,XQ11Gun\GunD:=XQ11GunData,XQ11GunTCP\Wobj:=wFM24B_Cabframe;
     SpotL wp429224,v2500,sd_wp429224,XQ11Gun\GunD:=XQ11GunData,XQ11GunTCP\Wobj:=wFM24B_Cabframe;
     SpotL wp429223,v2500,sd_wp429223,XQ11Gun\GunD:=XQ11GunData,XQ11GunTCP\Wobj:=wFM24B_Cabframe;
     MoveL Frwp429223_10,v2500,z50,XQ11GunTCP\Wobj:=wFM24B_Cabframe;
     MoveL Frwp429223_20,v2500,z50,XQ11GunTCP\Wobj:=wFM24B_Cabframe;
     MoveJ Frwp429223_30,v2500,z200,XQ11GunTCP\Wobj:=wFM24B_Cabframe;
     MoveJ Frwp429223_40,v2500,fine,XQ11GunTCP\Wobj:=wFM24B_Cabframe;
     RETURN;
  ENDPROC

  PROC FM24B_235_WSeg1()
     MoveAbsJ HomeXQ11Gun,v2500,fine,XQ11GunTCP;
     MoveJ Towp431451G_10,v2500,z200,XQ11GunTCP\Wobj:=wFM24B_Cabframe;
     MoveL Towp431451G_20,v2500,z50,XQ11GunTCP\Wobj:=wFM24B_Cabframe;
     SpotL wp431451G,v2500,sd_wp431451,XQ11Gun\GunD:=XQ11GunData,XQ11GunTCP\Wobj:=wFM24B_Cabframe;
     MoveL Towp431454_10,v2500,z50,XQ11GunTCP\Wobj:=wFM24B_Cabframe;
     MoveL Towp431454_20,v2500,z50,XQ11GunTCP\Wobj:=wFM24B_Cabframe;
     MoveJ Towp431454_30,v2500,z50,XQ11GunTCP\Wobj:=wFM24B_Cabframe;
     MoveJ Towp431454_40,v2500,z200,XQ11GunTCP\Wobj:=wFM24B_Cabframe;
     MoveL Towp431454_50,v2500,z50,XQ11GunTCP\Wobj:=wFM24B_Cabframe;
     MoveL Towp431454_60,v2500,z50,XQ11GunTCP\Wobj:=wFM24B_Cabframe;
     SpotL wp431454,v2500,sd_wp431454,XQ11Gun\GunD:=XQ11GunData,XQ11GunTCP\Wobj:=wFM24B_Cabframe;
     MoveL Towp431457_10,v2500,z50,XQ11GunTCP\Wobj:=wFM24B_Cabframe;
     MoveL Towp431457_20,v2500,z50,XQ11GunTCP\Wobj:=wFM24B_Cabframe;
     SpotL wp431457,v2500,sd_wp431457,XQ11Gun\GunD:=XQ11GunData,XQ11GunTCP\Wobj:=wFM24B_Cabframe;
     SpotL wp431458,v2500,sd_wp431458,XQ11Gun\GunD:=XQ11GunData,XQ11GunTCP\Wobj:=wFM24B_Cabframe;
     SpotL wp432845,v2500,sd_wp432845,XQ11Gun\GunD:=XQ11GunData,XQ11GunTCP\Wobj:=wFM24B_Cabframe;
     SpotL wp432844G,v2500,sd_wp432844,XQ11Gun\GunD:=XQ11GunData,XQ11GunTCP\Wobj:=wFM24B_Cabframe;
     SpotL wp431461,v2500,sd_wp431461,XQ11Gun\GunD:=XQ11GunData,XQ11GunTCP\Wobj:=wFM24B_Cabframe;
     SpotL wp431462,v2500,sd_wp431462,XQ11Gun\GunD:=XQ11GunData,XQ11GunTCP\Wobj:=wFM24B_Cabframe;
     SpotL wp431463,v2500,sd_wp431463,XQ11Gun\GunD:=XQ11GunData,XQ11GunTCP\Wobj:=wFM24B_Cabframe;
     SpotL wp431464,v2500,sd_wp431464,XQ11Gun\GunD:=XQ11GunData,XQ11GunTCP\Wobj:=wFM24B_Cabframe;
     MoveL Towp432811G_10,v2500,z50,XQ11GunTCP\Wobj:=wFM24B_Cabframe;
     MoveL Towp432811G_20,v2500,z50,XQ11GunTCP\Wobj:=wFM24B_Cabframe;
     MoveL Towp432811G_30,v2500,z50,XQ11GunTCP\Wobj:=wFM24B_Cabframe;
     SpotL wp432811G,v2500,sd_wp432811,XQ11Gun\GunD:=XQ11GunData,XQ11GunTCP\Wobj:=wFM24B_Cabframe;
     MoveL Towp432812G_10,v2500,z50,XQ11GunTCP\Wobj:=wFM24B_Cabframe;
     MoveL Towp432812G_20,v2500,z50,XQ11GunTCP\Wobj:=wFM24B_Cabframe;
     SpotL wp432812G,v2500,sd_wp432812,XQ11Gun\GunD:=XQ11GunData,XQ11GunTCP\Wobj:=wFM24B_Cabframe;
     MoveL Towp432815G_10,v2500,z50,XQ11GunTCP\Wobj:=wFM24B_Cabframe;
     MoveL Towp432815G_20,v2500,z50,XQ11GunTCP\Wobj:=wFM24B_Cabframe;
     MoveL Towp432815G_30,v2500,z50,XQ11GunTCP\Wobj:=wFM24B_Cabframe;
     MoveL Towp432815G_40,v2500,z50,XQ11GunTCP\Wobj:=wFM24B_Cabframe;
     MoveL Towp432815G_50,v2500,z50,XQ11GunTCP\Wobj:=wFM24B_Cabframe;
     SpotL wp432815G,v2500,sd_wp432815,XQ11Gun\GunD:=XQ11GunData,XQ11GunTCP\Wobj:=wFM24B_Cabframe;
     MoveL Towp432814G_10,v2500,z50,XQ11GunTCP\Wobj:=wFM24B_Cabframe;
     MoveL Towp432814G_20,v2500,z50,XQ11GunTCP\Wobj:=wFM24B_Cabframe;
     SpotL wp432814G,v2500,sd_wp432814,XQ11Gun\GunD:=XQ11GunData,XQ11GunTCP\Wobj:=wFM24B_Cabframe;
     MoveL Towp431473_10,v2500,z50,XQ11GunTCP\Wobj:=wFM24B_Cabframe;
     MoveL Towp431473_20,v2500,z50,XQ11GunTCP\Wobj:=wFM24B_Cabframe;
     SpotL wp431473,v2500,sd_wp431473,XQ11Gun\GunD:=XQ11GunData,XQ11GunTCP\Wobj:=wFM24B_Cabframe;
     SpotL wp431471,v2500,sd_wp431471,XQ11Gun\GunD:=XQ11GunData,XQ11GunTCP\Wobj:=wFM24B_Cabframe;
     SpotL wp431470,v2500,sd_wp431470,XQ11Gun\GunD:=XQ11GunData,XQ11GunTCP\Wobj:=wFM24B_Cabframe;
     SpotL wp431469,v2500,sd_wp431469,XQ11Gun\GunD:=XQ11GunData,XQ11GunTCP\Wobj:=wFM24B_Cabframe;
     MoveL Towp431468G_10,v2500,z50,XQ11GunTCP\Wobj:=wFM24B_Cabframe;
     MoveL Towp431468G_20,v2500,z50,XQ11GunTCP\Wobj:=wFM24B_Cabframe;
     SpotL wp431468G,v2500,sd_wp431468,XQ11Gun\GunD:=XQ11GunData,XQ11GunTCP\Wobj:=wFM24B_Cabframe;
     MoveL Frwp431468G_10,v2500,z50,XQ11GunTCP\Wobj:=wFM24B_Cabframe;
     MoveL Frwp431468G_20,v2500,z50,XQ11GunTCP\Wobj:=wFM24B_Cabframe;
     MoveL Frwp431468G_30,v2500,z50,XQ11GunTCP\Wobj:=wFM24B_Cabframe;
     MoveL Frwp431468G_40,v2500,z50,XQ11GunTCP\Wobj:=wFM24B_Cabframe;
     MoveJ Frwp431468G_50,v2500,fine,XQ11GunTCP\Wobj:=wFM24B_Cabframe;
     RETURN;
  ENDPROC

  PROC FM24B_14_WSeg2()
     MoveJ Towp433113_10,v2500,z200,XQ11GunTCP\Wobj:=wFM24BL1_CabframeGrip;
     MoveL Towp433113_20,v2500,z200,XQ11GunTCP\Wobj:=wFM24BL1_CabframeGrip;
     MoveL Towp433113_30,v2500,z50,XQ11GunTCP\Wobj:=wFM24BL1_CabframeGrip;
     SpotL wp433113,v2500,sd_wp433113,XQ11Gun\GunD:=XQ11GunData,XQ11GunTCP\Wobj:=wFM24BL1_CabframeGrip;
     SpotL wp433110,v2500,sd_wp433110,XQ11Gun\GunD:=XQ11GunData,XQ11GunTCP\Wobj:=wFM24BL1_CabframeGrip;
     RETURN;
  ENDPROC

  PROC FM24B_14_WSeg3()
     SpotL wp432852,v2500,sd_wp432852,XQ11Gun\GunD:=XQ11GunData,XQ11GunTCP\Wobj:=wFM24BL1_CabframeGrip;
     SpotL wp432849,v2500,sd_wp432849,XQ11Gun\GunD:=XQ11GunData,XQ11GunTCP\Wobj:=wFM24BL1_CabframeGrip;
     RETURN;
  ENDPROC

  PROC FM24B_14_WSeg4()
     MoveL Frwp432849_10,v2500,z50,XQ11GunTCP\Wobj:=wFM24BL1_CabframeGrip;
     MoveL Frwp432849_20,v2500,z50,XQ11GunTCP\Wobj:=wFM24BL1_CabframeGrip;
     MoveL Frwp432849_30,v2500,z50,XQ11GunTCP\Wobj:=wFM24BL1_CabframeGrip;
     MoveJ Frwp432849_50,v2500,z200,XQ11GunTCP\Wobj:=wFM24BL1_CabframeGrip;
     MoveJ Frwp432849_60,v2500,z200,XQ11GunTCP\Wobj:=wFM24BL1_CabframeGrip;
     MoveAbsJ HomeXQ11Gun,v2500,fine,XQ11GunTCP;
     RETURN;
  ENDPROC

  PROC FM24B_235_WSeg2()
     MoveJ Towp431452_20,v2500,z200,XQ11GunTCP\Wobj:=wFM24BL2_CabframeGrip;
     MoveL Towp431452_30,v2500,z50,XQ11GunTCP\Wobj:=wFM24BL2_CabframeGrip;
     SpotL wp431452,v2500,sd_wp431452,XQ11Gun\GunD:=XQ11GunData,XQ11GunTCP\Wobj:=wFM24BL2_CabframeGrip;
     SpotL wp431453,v2500,sd_wp431453,XQ11Gun\GunD:=XQ11GunData,XQ11GunTCP\Wobj:=wFM24BL2_CabframeGrip;
     MoveL Towp432847_10,v2500,z50,XQ11GunTCP\Wobj:=wFM24BL2_CabframeGrip;
     SpotL wp432847,v2500,sd_wp432847,XQ11Gun\GunD:=XQ11GunData,XQ11GunTCP\Wobj:=wFM24BL2_CabframeGrip;
     SpotL wp432846,v2500,sd_wp432846,XQ11Gun\GunD:=XQ11GunData,XQ11GunTCP\Wobj:=wFM24BL2_CabframeGrip;
     MoveL Towp431472_10,v2500,z50,XQ11GunTCP\Wobj:=wFM24BL2_CabframeGrip;
     MoveL Towp431472_20,v2500,z50,XQ11GunTCP\Wobj:=wFM24BL2_CabframeGrip;
     SpotL wp431472,v2500,sd_wp431472,XQ11Gun\GunD:=XQ11GunData,XQ11GunTCP\Wobj:=wFM24BL2_CabframeGrip;
     MoveL Towp432810_10,v2500,z50,XQ11GunTCP\Wobj:=wFM24BL2_CabframeGrip;
     MoveL Towp432810_20,v2500,z50,XQ11GunTCP\Wobj:=wFM24BL2_CabframeGrip;
     SpotL wp432810,v2500,sd_wp432810,XQ11Gun\GunD:=XQ11GunData,XQ11GunTCP\Wobj:=wFM24BL2_CabframeGrip;
     MoveL Frwp432810_10,v2500,z50,XQ11GunTCP\Wobj:=wFM24BL2_CabframeGrip;
     MoveL Frwp432810_20,v2500,z50,XQ11GunTCP\Wobj:=wFM24BL2_CabframeGrip;
     MoveJ Frwp432810_30,v2500,z200,XQ11GunTCP\Wobj:=wFM24BL2_CabframeGrip;
     MoveAbsJ HomeXQ11Gun,v2500,fine,XQ11GunTCP;
     RETURN;
  ENDPROC

ENDMODULE
